Staubli VAL3: writeStrValue.pgx

public program writeStrValue(num handle_, num col_, num row_, string value_, bool& result_[])
  local string strCell
begin
  // write a string value into a cell
  nCommand[handle_]=coSS
  call coord2Cell(col_,row_,strCell)
  call sendCommand(handle_,"ss"+strCell+value_,result_)
end
